RoboDK station: Stringer C-Corner-Top-Long-BOX2.rdk

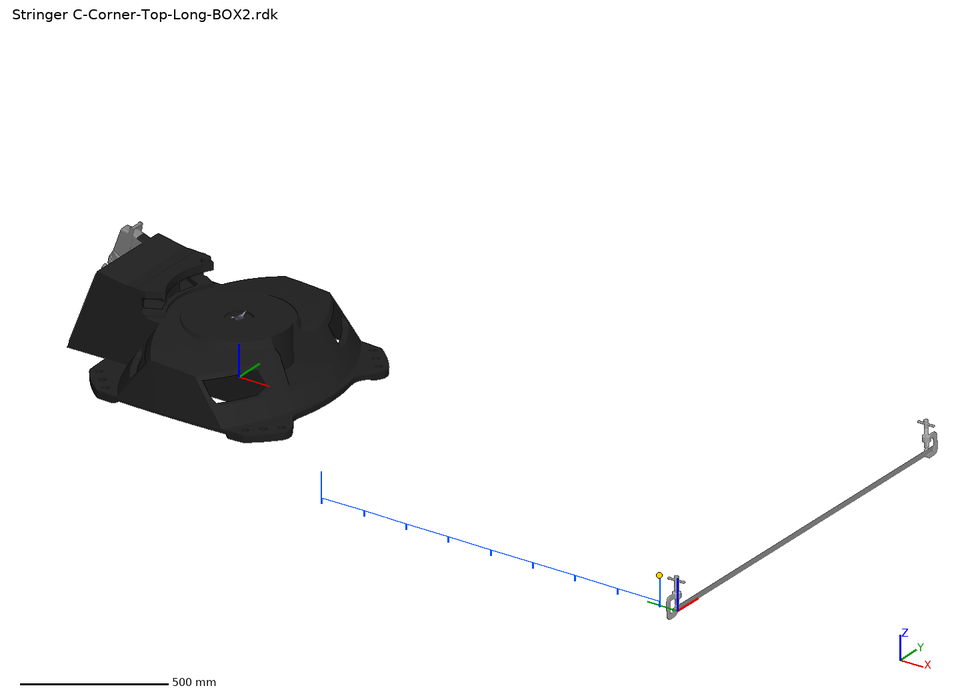
[picture v0: the station drawn from its stored meshes, robots at their saved joint values, targets as dots, program paths as lines]
Station Stringer C-Corner-Top-Long-BOX2 (saved by RoboDK 5.2.3). Poses are relative to the parent item; angles as X-Y-Z fixed-axis rotations.
  - frame KUKA KR 210 R2700 extra Base at (0, 0, 0) mm
    - robot KUKA KR 210 R2700 extra: 6 axes, payload 210 kg, reach 2696 mm, repeatability 0.06 mm, weight 1068 kg
        joint limits [-185, -140, -120, -350, -125, -350] to [185, -5, 155, 350, 125, 350]; home [0, -90, 90, 0, 0, 0]; saved at [-43.781, -22.764, 75.791, 76.517, 26.601, -111.667]
      - tool Spindle, TCP at (32, 0, 260) mm, rotated rx 0 ry 39 rz 0 deg, size 157.3 x 72 x 259.9 mm
  - frame Frame 2 at (1800, 0, -372.68) mm, rotated rx 0 ry 0 rz 90 deg
    - object L-Stringer C-top-corner -long- box2 at (0, 0, 0) mm, size 1499.5 x 20 x 20 mm, geometry from L-Stringer C-top-corner -long- box2.stl
    - object Stringer C-Corner-Top-Long-BOX2 at (0, 0, 0) mm, rotated rx 0 ry 0 rz -90 deg, 9 curves, geometry from Point 9
  - machining project Point settings: rotZ(0) | rotX(0)*rotY(0) | rotz(0) | onStart | onPathStart | onApproach | onPoint | onRetract | onFinish | SetRPM(%1) | SetTool(%1) | Extruder(%1) | default | default | OutOnMov(%1) | OutOffMov(%1) | onPathFinish | M_RunCode(%1)
  - program Point (56 instructions, listed below)
  - object FinalClamp at (1782.92, 1482.61, -312.65) mm, rotated rx 0 ry 88.65 rz 0 deg, size 145.3 x 71.1 x 72 mm, geometry from FinalClamp.stp
  - object FinalClamp2 at (1786.13, 14.22, -310.32) mm, rotated rx 177.11 ry 88.55 rz -2.31 deg, size 145.3 x 71.1 x 72 mm, geometry from FinalClamp.stp
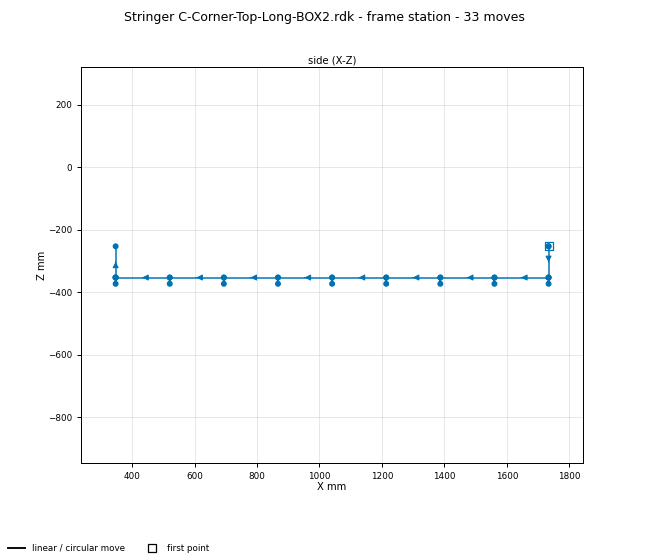
[picture p0: tool path of Stringer C-Corner-Top-Long-BOX2.rdk in frame station, 33 of 33 moves have a stored position in this frame; points joined in program order, loops and branches not executed]

--- program Point (robot KUKA KR 210 R2700 extra) ---
  Smooth(1)
  Set speed (1000.0 mm/s)
  Set Ref.: Frame 2
  Set Tool: Spindle
  Show Spindle
  MoveJ 1 to (-10.2, 66.57, 120) mm, rotated rx -180 ry 0 rz -180 deg; joints [-2.515, -34.002, 111.787, 176.489, 26.801, -178.82]
  MoveL 2 to (-10.2, 66.57, 120) mm, rotated rx -180 ry 0 rz -180 deg; joints [-2.515, -34.002, 111.787, 176.489, 26.801, -178.82]
  MoveL 3 to (-10.2, 66.57, 20) mm, rotated rx 180 ry 0 rz 180 deg; joints [-2.515, -28.676, 109.145, 176.784, 29.481, -179.154]
  MoveL 4 to (-10.2, 66.57, 20) mm, rotated rx 180 ry 0 rz 180 deg; joints [-2.515, -28.676, 109.145, 176.784, 29.481, -179.154]
  Set speed (50.0 mm/s)
  MoveL 5 to (-10.2, 66.57, 0) mm, rotated rx 180 ry 0 rz 180 deg; joints [-2.515, -27.618, 108.57, 176.831, 29.962, -179.208]
  MoveL 6 to (-10.2, 66.57, 20) mm, rotated rx 180 ry 0 rz 180 deg; joints [-2.515, -28.676, 109.145, 176.784, 29.481, -179.154]
  Set speed (1000.0 mm/s)
  MoveL 7 to (-10.2, 239.82, 20) mm, rotated rx 180 ry 0 rz -180 deg; joints [-8.991, -28.547, 108.238, 168.242, 28.856, -176.678]
  Set speed (50.0 mm/s)
  MoveL 8 to (-10.2, 239.82, 0) mm, rotated rx 180 ry 0 rz 180 deg; joints [-8.991, -27.498, 107.666, 168.415, 29.323, -176.876]
  MoveL 9 to (-10.2, 239.82, 20) mm, rotated rx 180 ry 0 rz -180 deg; joints [-8.991, -28.547, 108.238, 168.242, 28.856, -176.678]
  Set speed (1000.0 mm/s)
  MoveL 10 to (-10.2, 413.07, 20) mm, rotated rx -180 ry 0 rz -180 deg; joints [-15.244, -28.241, 106.313, 159.105, 27.642, -173.273]
  Set speed (50.0 mm/s)
  MoveL 11 to (-10.2, 413.07, 0) mm, rotated rx 180 ry 0 rz -180 deg; joints [-15.244, -27.209, 105.747, 159.418, 28.079, -173.627]
  MoveL 12 to (-10.2, 413.07, 20) mm, rotated rx -180 ry 0 rz -180 deg; joints [-15.244, -28.241, 106.313, 159.105, 27.642, -173.273]
  Set speed (1000.0 mm/s)
  MoveL 13 to (-10.2, 586.32, 20) mm, rotated rx -180 ry 0 rz -180 deg; joints [-21.147, -27.695, 103.382, 148.915, 26.087, -168.297]
  Set speed (50.0 mm/s)
  MoveL 14 to (-10.2, 586.32, 0) mm, rotated rx 180 ry 0 rz 180 deg; joints [-21.147, -26.687, 102.825, 149.384, 26.475, -168.82]
  MoveL 15 to (-10.2, 586.32, 20) mm, rotated rx -180 ry 0 rz -180 deg; joints [-21.147, -27.695, 103.382, 148.915, 26.087, -168.297]
  Set speed (1000.0 mm/s)
  MoveL 16 to (-10.2, 759.57, 20) mm, rotated rx 180 ry 0 rz -180 deg; joints [-26.616, -26.832, 99.457, 137.238, 24.536, -161.205]
  Set speed (50.0 mm/s)
  MoveL 17 to (-10.2, 759.57, 0) mm, rotated rx 180 ry 0 rz 180 deg; joints [-26.616, -25.852, 98.908, 137.871, 24.854, -161.902]
  MoveL 18 to (-10.2, 759.57, 20) mm, rotated rx 180 ry 0 rz -180 deg; joints [-26.616, -26.832, 99.457, 137.238, 24.536, -161.205]
  Set speed (1000.0 mm/s)
  MoveL 19 to (-10.2, 932.82, 20) mm, rotated rx -180 ry 0 rz -180 deg; joints [-31.609, -25.57, 94.537, 123.862, 23.404, -151.734]
  Set speed (50.0 mm/s)
  MoveL 20 to (-10.2, 932.82, 0) mm, rotated rx 180 ry 0 rz 180 deg; joints [-31.609, -24.622, 93.996, 124.635, 23.633, -152.577]
  MoveL 21 to (-10.2, 932.82, 20) mm, rotated rx -180 ry 0 rz -180 deg; joints [-31.609, -25.57, 94.537, 123.862, 23.404, -151.734]
  Set speed (1000.0 mm/s)
  MoveL 22 to (-10.2, 1106.07, 20) mm, rotated rx 180 ry 0 rz 180 deg; joints [-36.119, -23.828, 88.598, 109.119, 23.118, -140.21]
  Set speed (50.0 mm/s)
  MoveL 23 to (-10.2, 1106.07, 0) mm, rotated rx 180 ry 0 rz 180 deg; joints [-36.119, -22.912, 88.06, 109.953, 23.244, -141.117]
  MoveL 24 to (-10.2, 1106.07, 20) mm, rotated rx 180 ry 0 rz 180 deg; joints [-36.119, -23.828, 88.598, 109.119, 23.118, -140.21]
  Set speed (1000.0 mm/s)
  MoveL 25 to (-10.2, 1279.32, 20) mm, rotated rx 180 ry 0 rz -180 deg; joints [-40.165, -21.517, 81.565, 94.041, 24.011, -127.684]
  Set speed (50.0 mm/s)
  MoveL 26 to (-10.2, 1279.32, 0) mm, rotated rx -180 ry 0 rz 180 deg; joints [-40.165, -20.63, 81.023, 94.814, 24.038, -128.531]
  MoveL 27 to (-10.2, 1279.32, 20) mm, rotated rx 180 ry 0 rz -180 deg; joints [-40.165, -21.517, 81.565, 94.041, 24.011, -127.684]
  Set speed (1000.0 mm/s)
  MoveL 28 to (-10.2, 1452.57, 20) mm, rotated rx -180 ry 0 rz 180 deg; joints [-43.781, -18.522, 73.28, 79.927, 26.247, -115.474]
  Set speed (50.0 mm/s)
  MoveL 29 to (-10.2, 1452.57, 0) mm, rotated rx 180 ry 0 rz 180 deg; joints [-43.781, -17.658, 72.723, 80.541, 26.195, -116.158]
  MoveL 30 to (-10.2, 1452.57, 20) mm, rotated rx -180 ry 0 rz 180 deg; joints [-43.781, -18.522, 73.28, 79.927, 26.247, -115.474]
  MoveL 31 to (-10.2, 1452.57, 20) mm, rotated rx -180 ry 0 rz 180 deg; joints [-43.781, -18.522, 73.28, 79.927, 26.247, -115.474]
  Set speed (1000.0 mm/s)
  MoveL 32 to (-10.2, 1452.57, 20) mm, rotated rx -180 ry 0 rz 180 deg; joints [-43.781, -18.522, 73.28, 79.927, 26.247, -115.474]
  MoveL 33 to (-10.2, 1452.57, 120) mm, rotated rx -180 ry 0 rz 180 deg; joints [-43.781, -22.764, 75.791, 76.517, 26.601, -111.667]
